// Mitsubishi GX Works2 project: z08   PLC: Q02/Q02H

PROGRAM MAIN
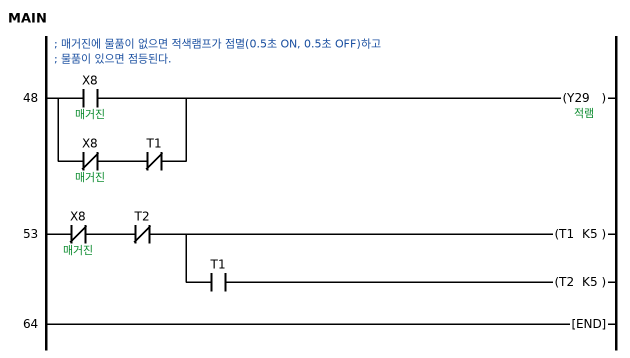
; 매거진에 물품이 없으면 적색램프가 점멸(0.5초 ON, 0.5초 OFF)하고
; 물품이 있으면 점등된다.
48    LD      X8  ; 매거진
      LDI     X8  ; 매거진
      ANI     T1
      ORB
      OUT     Y29  ; 적램
53    LDI     X8  ; 매거진
      ANI     T2
      OUT     T1 K5
      AND     T1
      OUT     T2 K5
64    END
END_PROGRAM

// device comments not shown above
X0  ; 공급_후
X1  ; 공급_전
X2  ; 드릴_상
X3  ; 드릴_하
X4  ; 송출_후
X5  ; 송출_전
X6  ; 배출_후
X7  ; 배출_전
X9  ; 이송감지
X0A  ; 비금속
X0B  ; 금속
X0C  ; PB1
X0D  ; PB2
X0E  ; PB3
X0F  ; 비상정지
Y20  ; 공급_전
Y21  ; 공급_후
Y22  ; 드릴_실
Y23  ; 송출_전
Y24  ; 송출_후
Y25  ; 배출_전
Y26  ; 배출_후
Y27  ; 드릴_모
Y28  ; 컨베
Y2A  ; 황램
Y2B  ; 녹램
